PROGRAM MAIN_CFC
VAR
	Timer			: TON;
	fbCFC_SamplePOU : FB_CFC_SamplePOU;

	eOperation		: E_Operation := eOp_Add;
	eOperationPrev	: E_Operation := eOp_Add;
	iResultC		: DINT;
	bZero			: BOOL;
	bPos			: BOOL;
	bNeg			: BOOL;
	bTest			: BOOL;
	tTimerValue		: TIME := T#3S;
END_VAR
VAR // added by the converter: edge detectors and wires of the graphical bodies
    _w1, _w2, _w3 : E_Operation;
END_VAR

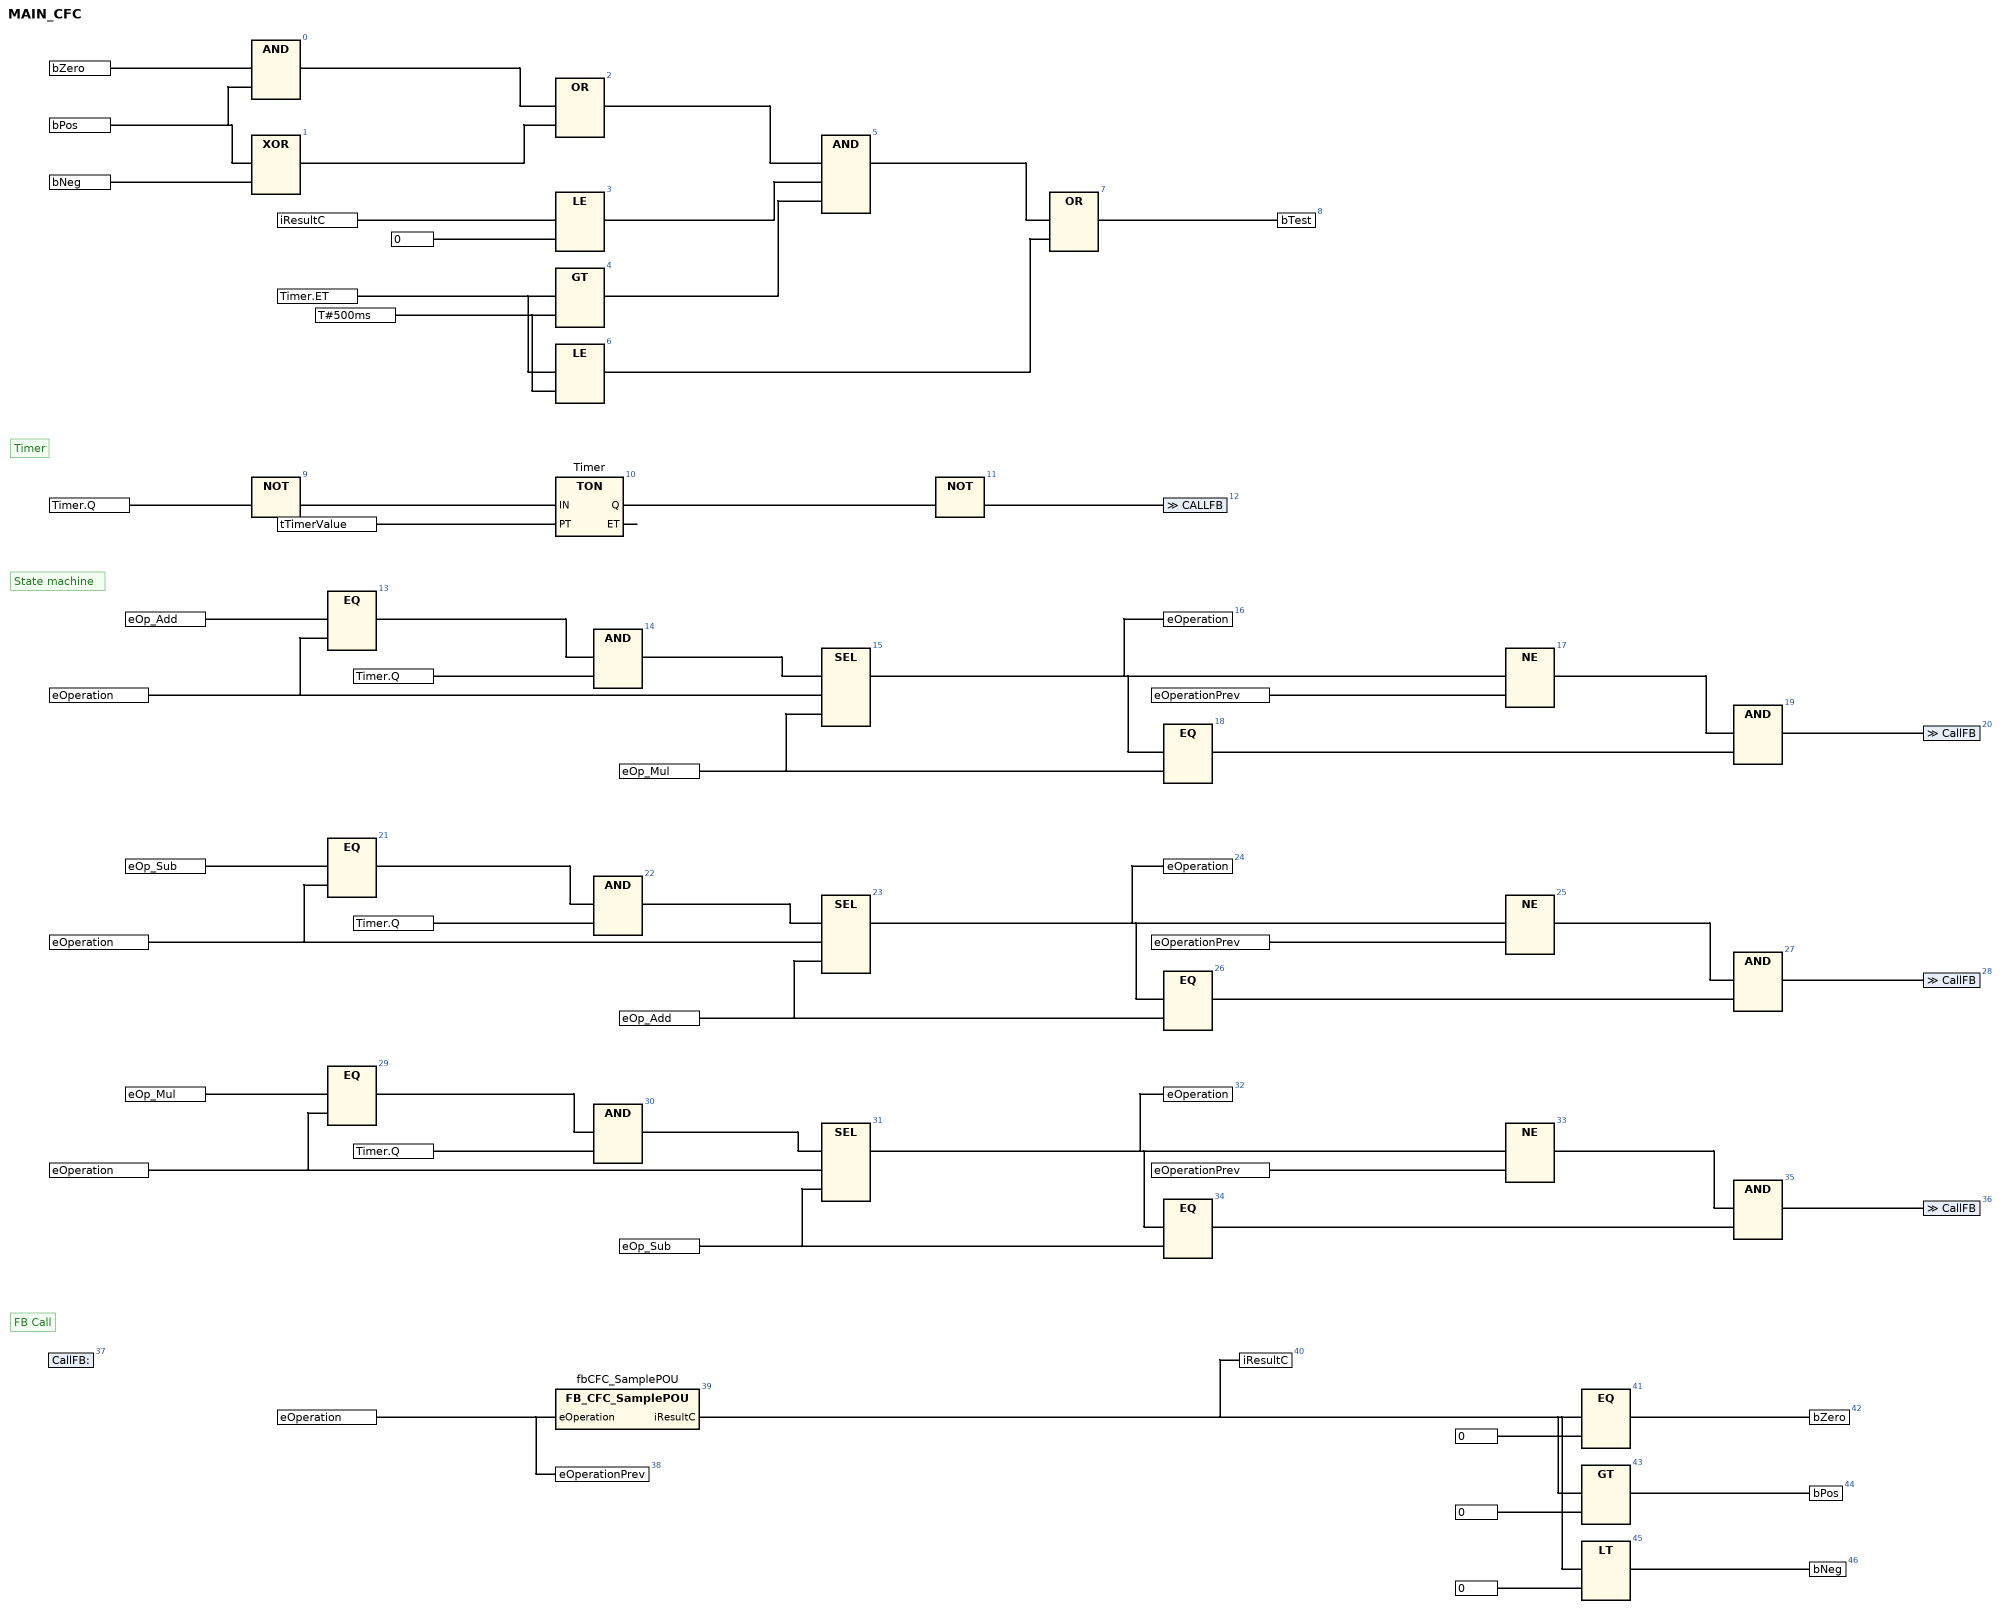
bTest := (bZero AND bPos OR bPos XOR bNeg) AND iResultC <= 0 AND Timer.ET > T#500ms OR Timer.ET <= T#500ms;
// Timer
Timer(IN := NOT Timer.Q, PT := tTimerValue); // TON
IF NOT Timer.Q THEN JMP CALLFB; END_IF
// State machine
_w1 := SEL(eOp_Add = eOperation AND Timer.Q, eOperation, eOp_Mul);
eOperation := _w1;
IF _w1 <> eOperationPrev AND _w1 = eOp_Mul THEN JMP CallFB; END_IF
_w2 := SEL(eOp_Sub = eOperation AND Timer.Q, eOperation, eOp_Add);
eOperation := _w2;
IF _w2 <> eOperationPrev AND _w2 = eOp_Add THEN JMP CallFB; END_IF
_w3 := SEL(eOp_Mul = eOperation AND Timer.Q, eOperation, eOp_Sub);
eOperation := _w3;
IF _w3 <> eOperationPrev AND _w3 = eOp_Sub THEN JMP CallFB; END_IF
// FB Call
CallFB: ;
eOperationPrev := eOperation;
fbCFC_SamplePOU(eOperation := eOperation); // FB_CFC_SamplePOU
iResultC := fbCFC_SamplePOU.iResultC;
bZero := fbCFC_SamplePOU.iResultC = 0;
bPos := fbCFC_SamplePOU.iResultC > 0;
bNeg := fbCFC_SamplePOU.iResultC < 0;

END_PROGRAM

(* stored: Version 1.1.0.1, ProductVersion 3.1.4024.11
   POU MAIN_CFC: Id {285bbb03-3e2b-44dc-ab09-36066decee31}, SpecialFunc None *)
